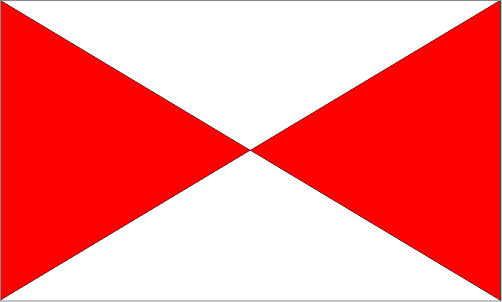
VISUALIZATION visuHSVSim  // 502x302
    Group (0,0 500x300)
        Polygon (0,0) (0,300) (250,150), invisible if: NOT progHSVCntrl.HSV_04_0100.FB_Close
        Polygon (500,0) (500,300) (250,150), invisible if: NOT progHSVCntrl.HSV_04_0100.FB_Close
        Polygon (0,0) (0,300) (250,150), invisible if: NOT progHSVCntrl.HSV_04_0100.FB_Travelling
        Polygon (500,0) (500,300) (250,150), invisible if: NOT progHSVCntrl.HSV_04_0100.FB_Travelling
        Polygon (0,0) (0,300) (250,150), invisible if: NOT progHSVCntrl.HSV_04_0100.FB_Open
        Polygon (500,0) (500,300) (250,150), invisible if: NOT progHSVCntrl.HSV_04_0100.FB_Open
        Polygon (0,0) (0,300) (250,150), invisible if: NOT progHSVCntrl.HSV_04_0100.Alarm
        Polygon (500,0) (500,300) (250,150), invisible if: NOT progHSVCntrl.HSV_04_0100.Alarm
END_VISUALIZATION

(* stored: Version 1.1.0.1, ProductVersion 3.1.4022.17
   Visu visuHSVSim: Id {5ca31e3b-2f57-4dc3-a0ad-d989e833ef70} *)
